// TIA Portal project "ControlCintas" (V16)

(* hardware
DEVICE "S7-1200 station_1"  S7-1200 Station
   slot 0: "Rack_0"  S7-1200 Rack  Rack  V1.0
   slot 1: "PLC_1"  CPU 1214C DC/DC/DC  6ES7 214-1AG40-0XB0  V4.4
   slot 2: "AI 4xRTD_1"  6ES7 231-5PD30-0XB0  V1.0
   slot 3: "AQ 4x14BIT_1"  SM 1232 AQ4  6ES7 232-4HD30-0XB0  V1.0
*)

// ===== PLC "PLC_1"  CPU 1214C DC/DC/DC =====

VAR_GLOBAL   // PLC tag table "Tabla de variables estándar"
   "Motor Cinta 1" AT %Q0.0 : Bool;
   "Motor Cinta 2" AT %Q0.1 : Bool;
   "Motor Cinta 3" AT %Q0.2 : Bool;
   "Start Cinta 1" AT %I0.0 : Bool;
   "Start Cinta 2" AT %I0.1 : Bool;
   "Start Cinta 3" AT %I0.2 : Bool;
   "Sensor Cinta 1" AT %I0.3 : Bool;
   "Sensor Cinta 2" AT %I0.4 : Bool;
   "Sensor Cinta 3" AT %I0.5 : Bool;
   "Emergencia" AT %I1.1 : Bool;
   "DISCONNECT" AT %M0.0 : Bool;
END_VAR

DATA_BLOCK "ControlCintas"   // DB1
{ S7_Optimized_Access := 'FALSE' }
VERSION : 0.1
   VAR
      Cinta1_On : Bool;
      Cinta2_On : Bool;
      Cinta3_On : Bool;
   END_VAR
BEGIN
END_DATA_BLOCK

DATA_BLOCK "ControlAnalogicas"   // DB2
{ S7_Optimized_Access := 'TRUE' }
VERSION : 0.1
   VAR
      AI1 : Word;   // Valor de entrada analogica 1
      AI2 : Word;   // Valor de entrada analogica 2
      AI3 : Word;   // Valor de entrada analogica 3
      AI4 : Word;   // Valor de entrada analogica 4
      AI1_Scaled : Real;
      AI2_Scaled : Real;
      AI3_Scaled : Real;
      AI4_Scaled : Real;
      AQ1_Set : Real;
      AQ2_Set : Real;
      AQ3_Set : Real;
      AQ4_set : Real;
      AQ1_Set_Raw : Real;
      AQ2_Set_Raw : Real;
      AQ3_Set_Raw : Real;
      AQ4_Set_Raw : Real;
      ErrorDiagnostico : Bool;
   END_VAR
BEGIN
END_DATA_BLOCK

FUNCTION "FC_ScaleAnalog" : Void   // FC1, LAD
{ S7_Optimized_Access := 'TRUE' }
VERSION : 0.1
BEGIN

REGION Network 1
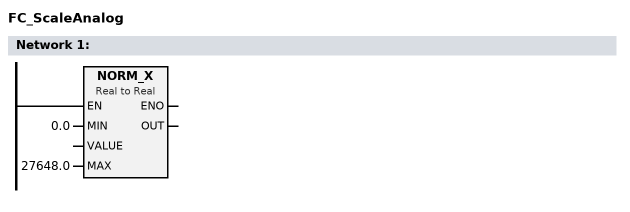
   RUNG wire#powerrail
      { S7_Templates := "[SrcType := Real, DestType := Real]" } Normalize(min := 0.0, value :=, max := 27648.0, out =>)
   END_RUNG
   // the same network as SCL:
   <??.?> := NORM_X(MIN := 0.0, MAX := 27648.0);
END_REGION
END_FUNCTION

ORGANIZATION_BLOCK "Main"   // OB1, LAD, ProgramCycle
TITLE = "Main Program Sweep (Cycle)"
{ S7_Optimized_Access := 'TRUE' }
VERSION : 0.1
BEGIN

REGION Network 1
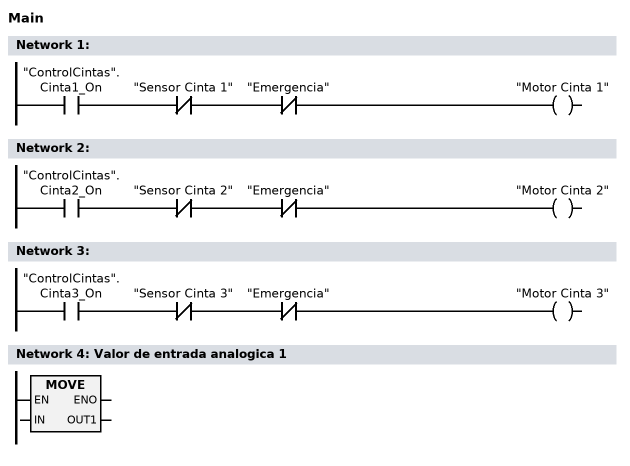
   RUNG wire#powerrail
      Contact( "ControlCintas".Cinta1_On )
      I_Contact( "Sensor Cinta 1" )
      I_Contact( "Emergencia" )
      Coil( "Motor Cinta 1" )
   END_RUNG
   // the same network as SCL:
   "Motor Cinta 1" := "ControlCintas".Cinta1_On AND NOT "Sensor Cinta 1" AND NOT "Emergencia";
END_REGION

REGION Network 2
   RUNG wire#powerrail
      Contact( "ControlCintas".Cinta2_On )
      I_Contact( "Sensor Cinta 2" )
      I_Contact( "Emergencia" )
      Coil( "Motor Cinta 2" )
   END_RUNG
   // the same network as SCL:
   "Motor Cinta 2" := "ControlCintas".Cinta2_On AND NOT "Sensor Cinta 2" AND NOT "Emergencia";
END_REGION

REGION Network 3
   RUNG wire#powerrail
      Contact( "ControlCintas".Cinta3_On )
      I_Contact( "Sensor Cinta 3" )
      I_Contact( "Emergencia" )
      Coil( "Motor Cinta 3" )
   END_RUNG
   // the same network as SCL:
   "Motor Cinta 3" := "ControlCintas".Cinta3_On AND NOT "Sensor Cinta 3" AND NOT "Emergencia";
END_REGION

REGION Network 4: Valor de entrada analogica 1
   RUNG wire#powerrail
      Move(in :=, out1 =>)
   END_RUNG
   // the same network as SCL:
   // no SCL statement known for Move: written as a call
   Move();
END_REGION
END_ORGANIZATION_BLOCK